TYPE stackerLoadSettings :
STRUCT
	
	axisLength                :   REAL   := 600; 		   // макс ход на оста на стакера за модел HEX 24
	axisWorkSpeed             :	  REAL   := 1000.0; 	   // скорост 
	axisInitSpeed			  :   REAL   := 2000.0; 	   // скорост при движение нагоре (при init)
	axisAcc					  :   REAL   := 0.2 ;          // ускр.
	palletSize                :   ARRAY[1..Consts.MAX_RECIPE] OF REAL; 

END_STRUCT
END_TYPE

(* stored: Version 1.1.0.1, ProductVersion 3.1.4024.3
   DUT stackerLoadSettings: Id {4d6720e7-4404-4a67-8f80-d50afb3160af} *)
